Omron Sysmac Studio project RemoteLab (Sysmac Studio 1.47.0.64008, StandardProject)

# Controller Controller_0: NJ301-1100 version 1.20
Units and slaves: Power Supply : NJ-Px3001; CPU : NJ301-1100; 0 : CJ1W-ID211 (J01); 1 : CJ1W-OC211 (J02)
Task PrimaryTask (priority 4, period or condition 4000): PrimaryTask_Main
Task CommTask (priority 16, period or condition 100000): CommTask_ModbusServer
Task ControlTask (priority 16, period or condition 40000): ControlTask_PID
Library MTCP_Server_NJNX 2.6. (contents left out)
Library MTCP_Client_NJ 2.6. (contents left out)

VAR_GLOBAL
    G_Eff_Mode : INT;
    G_Eff_PLC_Enable : BOOL;
    G_Eff_Setpoint : REAL;
    G_Eff_Manual_MV : REAL;
    G_Eff_StartAT : BOOL;
    G_Modbus_ReadBuf : ARRAY[0..1023] OF WORD;  (* Raw Read Data *)
    G_Modbus_WriteBuf : ARRAY[0..1023] OF WORD;  (* Raw Write Data (Mirror of Gateway HRs) *)
    G_OverheatLatched : BOOL;
    StartServer : BOOL := True;
    G_RTD_Temp : REAL;
    G_Setpoint : REAL := 0.0;
    G_StartAT : INT := 0;
    G_ATDone : WORD;
    G_Web_Status : INT := 0;  (* written by CommTask from HR3 *)
    G_Current_MV : REAL;
    G_Manual_MV : REAL := 0.0;  (* Extracted Manual MV *)
    G_Mode : INT := 0;  (* 0=Manual, 1=Auto, 2=Tune *)
    G_PID_PB : REAL;
END_VAR
VAR_GLOBAL RETAIN
    G_PID_PB_Out : REAL := 8.8;
END_VAR
VAR_GLOBAL
    G_PID_Td : REAL;
END_VAR
VAR_GLOBAL RETAIN
    G_PID_Td_Out : REAL := 50;
END_VAR
VAR_GLOBAL
    G_PID_Ti : REAL;
    HMI_AT_ON_Rise : BOOL;
    HMI_AT_OFF_Rise : BOOL;
    HMI_AT_ON_Prev : BOOL;
    HMI_AT_OFF_Prev : BOOL;
END_VAR
VAR_GLOBAL RETAIN
    G_PID_Ti_Out : REAL := 140;
END_VAR
VAR_GLOBAL
    G_PLC_Status : INT := 0;
    Heartbeat_Ctr : UINT;
    G_CommAlive : BOOL;  (* written by PrimaryTask (watchdog) *)
    HMI_Mode : INT;
    HMI_PLC_Enable : BOOL;  (* Momentary button to apply changes *)
    HMI_Setpoint : REAL;
    HMI_Manual_MV : REAL;
    HMI_AT_ON : BOOL;  (* Momentary pushbutton — Start Auto-Tune *)
    HMI_AT_OFF : BOOL;  (* Momentary pushbutton — Stop Auto-Tune *)
    HMI_StartAT : BOOL;
    Out_0 : BOOL;  (* Green LED; at IOBus://rack#0/slot#1/Ch1_Out/Ch1_Out00 *)
    Out_1 : BOOL;  (* Yellow LED; at IOBus://rack#0/slot#1/Ch1_Out/Ch1_Out01 *)
    Out_2 : BOOL;  (* RED LED; at IOBus://rack#0/slot#1/Ch1_Out/Ch1_Out02 *)
    Out_3 : BOOL;  (* PWM output to heater driver; at IOBus://rack#0/slot#1/Ch1_Out/Ch1_Out03 *)
    G_ATBusy : WORD;
    G_Tune_Err : WORD;
    G_WebActive : BOOL;
    HMI_PID_PB : REAL;  (* Proportional Band *)
    HMI_PID_Ti : REAL;  (* Integral Time (seconds) *)
    HMI_PID_Td : REAL;  (* Derivative Time (seconds) *)
    HMI_PID_Update : BOOL;
    HMI_PID_Update_Rise : BOOL;
    HMI_PID_Update_Prev : BOOL;
    HMI_PID_Update_Feedback : BOOL;  (* momentary indicator that tells the operator "Your parameters were successfully applied!" *)
    G_Eff_PID_PB : REAL;
    G_Eff_PID_Ti : REAL;
    G_Eff_PID_Td : REAL;
    C_MODE_MANUAL : INT := 0;
    C_MODE_AUTO : INT := 1;
    C_MODE_TUNE : INT := 2;
    HMI_Manual_MV_DataEdit : REAL;
    HMI_Setpoint_DataEdit : REAL;
    G_Mode_Manual : BOOL;
    G_Mode_AT : BOOL;
    G_Mode_Auto : BOOL;
    HMI_Manual_Start_Rise : BOOL;
    HMI_Manual_Start_Prev : BOOL;
    HMI_Manual_Start : BOOL;
    HMI_Manual_Stop : BOOL;
    HMI_Manual_Stop_Rise : BOOL;
    HMI_Manual_Stop_Prev : BOOL;
    G_PID_PB_AT : REAL;
    G_PID_Ti_AT : REAL;
    G_PID_Td_AT : REAL;
    HMI_Automatic_Start : BOOL;
    HMI_Automatic_Start_Rise : BOOL;
    HMI_Automatic_Start_Prev : BOOL;
    HMI_Automatic_Stop : BOOL;
    HMI_Automatic_Stop_Rise : BOOL;
    HMI_Automatic_Stop_Prev : BOOL;
    G_Heater_Power_W : REAL;
    G_ATDone_FB : BOOL;
END_VAR

PROGRAM CommTask_ModbusServer
VAR
    MB_Server : MTCP_Server_NJNX;
    Local_TcpPort : UINT := 1502;
    ConnectionTimeout : TIME := T#0ms;
    Reset_SdRcvCounter : BOOL := False;
    Server_Connected : BOOL;
    Server_Error : BOOL;
    Server_ErrorID : WORD;
    IP_Client : STRING[15];
    Port_Client : UINT;
    SdRcv_Counter : UDINT;
    SdRcv_Last : UDINT;
    Coils : ARRAY[0..1023] OF BOOL;
    Registers : ARRAY[0..1023] OF WORD;
    i : INT;
    New_Seq : WORD;
    Last_Seq_Num : WORD;
    R2W_MV : FB_RealToWords;
    R2W_PB : FB_RealToWords;
    R2W_Ti : FB_RealToWords;
    R2W_Td : FB_RealToWords;
    R2W_Setpoint : FB_RealToWords;
    R2W_PB_AT : FB_RealToWords;
    R2W_Ti_AT : FB_RealToWords;
    R2W_Td_AT : FB_RealToWords;
END_VAR
VAR_EXTERNAL
    G_Modbus_ReadBuf : ARRAY[0..1023] OF WORD;
    StartServer : BOOL;
    G_Web_Status : INT;
    G_Mode : INT;
    G_PLC_Status : INT;
    G_Manual_MV : REAL;
    G_Setpoint : REAL;
    G_StartAT : INT;
    G_PID_PB : REAL;
    G_PID_Ti : REAL;
    G_PID_Td : REAL;
    G_Current_MV : REAL;
    G_PID_Td_Out : REAL;
    G_Modbus_WriteBuf : ARRAY[0..1023] OF WORD;
    G_RTD_Temp : REAL;
    G_PID_PB_Out : REAL;
    G_PID_Ti_Out : REAL;
    Heartbeat_Ctr : UINT;
    G_ATDone : WORD;
    G_Eff_Setpoint : REAL;
    G_PID_PB_AT : REAL;
    G_PID_Ti_AT : REAL;
    G_PID_Td_AT : REAL;
    G_ATBusy : WORD;
    G_ATDone_FB : BOOL;
    G_Tune_Err : WORD;
END_VAR
(*
    CommTask_ModbusServer
    - PLC is Modbus TCP SERVER (slave)
    - Gateway/Web is Modbus TCP CLIENT (master)
*)

// =========================================================
// 1) Run the Modbus TCP Server FB EVERY scan
// =========================================================
MB_Server(
    Start             := StartServer,
    Local_TcpPort     := Local_TcpPort,
    ConnectionTimeout := ConnectionTimeout,
    Reset_SdRcvCounter:= Reset_SdRcvCounter,

    Registers         := Registers,
    Coils             := Coils,

    Connected         => Server_Connected,
    Error             => Server_Error,
    ErrorID           => Server_ErrorID,
    IP_Client         => IP_Client,
    Port_Client       => Port_Client,
    SdRcv_Counter     => SdRcv_Counter
);


// =========================================================
// 2) Heartbeat: increment when a Modbus transaction happened
//    (so it tracks real comm activity)
// =========================================================
IF SdRcv_Counter <> SdRcv_Last THEN
    SdRcv_Last := SdRcv_Counter;
    Heartbeat_Ctr := Heartbeat_Ctr + 1;
END_IF;


// =========================================================
// 3) Copy incoming gateway-written registers into your buffer
//    (HR0..HR16 -> G_Modbus_ReadBuf[0..16])
// =========================================================
FOR i := 0 TO 16 DO
    G_Modbus_ReadBuf[i] := Registers[i];
END_FOR;


// =========================================================
// 4) PROCESS (same as your old State 20)
// =========================================================
G_RTD_Temp := FUN_WordsToReal(G_Modbus_ReadBuf[1], G_Modbus_ReadBuf[2]);

New_Seq := G_Modbus_ReadBuf[0];

IF New_Seq <> Last_Seq_Num THEN
    G_Web_Status := WORD_TO_INT(G_Modbus_ReadBuf[3]);
    G_Mode       := WORD_TO_INT(G_Modbus_ReadBuf[4]);
    G_PLC_Status := WORD_TO_INT(G_Modbus_ReadBuf[5]);

    G_Manual_MV  := FUN_WordsToReal(G_Modbus_ReadBuf[6], G_Modbus_ReadBuf[7]);
    G_Setpoint   := FUN_WordsToReal(G_Modbus_ReadBuf[8], G_Modbus_ReadBuf[9]);

    G_StartAT   := WORD_TO_INT(G_Modbus_ReadBuf[10]);

    G_PID_PB     := FUN_WordsToReal(G_Modbus_ReadBuf[11], G_Modbus_ReadBuf[12]);
    G_PID_Ti     := FUN_WordsToReal(G_Modbus_ReadBuf[13], G_Modbus_ReadBuf[14]);
    G_PID_Td     := FUN_WordsToReal(G_Modbus_ReadBuf[15], G_Modbus_ReadBuf[16]);

    Last_Seq_Num := New_Seq;
END_IF;


// =========================================================
// 5) BUILD WRITE BUFFER (same as your old State 30)
//    (HR100..HR110 -> G_Modbus_WriteBuf[0..10])
// =========================================================
G_Modbus_WriteBuf[0] := Last_Seq_Num;                // HR100 ack seq
G_Modbus_WriteBuf[1] := UINT_TO_WORD(Heartbeat_Ctr); // HR101 heartbeat

R2W_MV(InReal := G_Current_MV);
G_Modbus_WriteBuf[2] := R2W_MV.W_High;               // HR102  -- Current_MV
G_Modbus_WriteBuf[3] := R2W_MV.W_Low;                // HR103

// ===== Autotune Status =====
G_Modbus_WriteBuf[4] := G_ATBusy;        // HR104  autotune running
G_Modbus_WriteBuf[5] := G_ATDone;     // HR105  autotune finished
G_Modbus_WriteBuf[6] := G_Tune_Err;      // HR106  autotune error

// ===== Current PID parameters =====
R2W_PB(InReal := G_PID_PB_Out);
G_Modbus_WriteBuf[7] := R2W_PB.W_High;               // HR107
G_Modbus_WriteBuf[8] := R2W_PB.W_Low;                // HR108

R2W_Ti(InReal := G_PID_Ti_Out);
G_Modbus_WriteBuf[9]  := R2W_Ti.W_High;              // HR109
G_Modbus_WriteBuf[10] := R2W_Ti.W_Low;               // HR110

R2W_Td(InReal := G_PID_Td_Out);
G_Modbus_WriteBuf[11] := R2W_Td.W_High;              // HR111
G_Modbus_WriteBuf[12] := R2W_Td.W_Low;               // HR112

// ===== Current Setpoint =====
R2W_Setpoint(InReal := G_Eff_Setpoint);
G_Modbus_WriteBuf[13] := R2W_Setpoint.W_High;        // HR113
G_Modbus_WriteBuf[14] := R2W_Setpoint.W_Low;         // HR114

// ===== Autotune Results =====
R2W_PB_AT(InReal := G_PID_PB_AT);
G_Modbus_WriteBuf[15] := R2W_PB_AT.W_High;           // HR115
G_Modbus_WriteBuf[16] := R2W_PB_AT.W_Low;            // HR116

R2W_Ti_AT(InReal := G_PID_Ti_AT);
G_Modbus_WriteBuf[17] := R2W_Ti_AT.W_High;           // HR117
G_Modbus_WriteBuf[18] := R2W_Ti_AT.W_Low;            // HR118

R2W_Td_AT(InReal := G_PID_Td_AT);
G_Modbus_WriteBuf[19] := R2W_Td_AT.W_High;           // HR119
G_Modbus_WriteBuf[20] := R2W_Td_AT.W_Low;            // HR120

// =========================================================
// 6) Copy your write buffer into server registers
//    (G_Modbus_WriteBuf -> HR100..HR110)
// =========================================================
FOR i := 0 TO 20 DO
    Registers[100 + i] := G_Modbus_WriteBuf[i];
END_FOR;
END_PROGRAM

PROGRAM ControlTask_PID
VAR
    ATBusy_FB : BOOL;
    ATErr_FB : BOOL;
    ATErrID_FB : WORD;
    TuneCmd : BOOL;
    Ti_ms : DINT;
    Td_ms : DINT;
    Ti_Time : TIME;
    Td_Time : TIME;
    StartAT_Cmd : BOOL;
    RunCmd : BOOL;
    MV_fromPID : REAL;
    MV_percent : REAL;
    OprSetParams : _sOPR_SET_PARAMS := (MVLowLmt := 0.0, MVUpLmt := 100.0, ManResetVal := 0.0, MVTrackSw := False, MVTrackVal := 0.0, StopMV := 0.0, ErrorMV := 0.0, Alpha := 0.0, ATCalcGain := 1.0, ATHystrs := 0.2);
    InitSetParams : _sINIT_SET_PARAMS := (SampTime := T#200mS, RngLowLmt := 0.0, RngUpLmt := 150.0, DirOpr := False);
    PB_Active : REAL;
    Ti_Active_s : REAL;
    Td_Active_s : REAL;
    Ti_Active : REAL;
    Td_Active : REAL;
    PIDAT_instance : PIDAT;
    ATDone_Rise : BOOL;
    ATDone_Prev : BOOL;
END_VAR
VAR_EXTERNAL
    G_Eff_Mode : INT;
    G_PID_PB : REAL;
    G_PID_Ti : REAL;
    G_PID_Td : REAL;
    G_PID_PB_Out : REAL;
    G_PID_Ti_Out : REAL;
    G_PID_Td_Out : REAL;
    G_Eff_PLC_Enable : BOOL;
    G_OverheatLatched : BOOL;
    G_Eff_StartAT : BOOL;
    G_RTD_Temp : REAL;
    G_Eff_Setpoint : REAL;
    G_Eff_Manual_MV : REAL;
    G_Current_MV : REAL;
    G_ATBusy : WORD;
    G_Tune_Err : WORD;
    G_ATDone : WORD;
    G_WebActive : BOOL;
    HMI_PID_PB : REAL;
    HMI_PID_Ti : REAL;
    HMI_PID_Td : REAL;
    HMI_PID_Update_Rise : BOOL;
    HMI_PID_Update : BOOL;
    HMI_PID_Update_Prev : BOOL;
    HMI_PID_Update_Feedback : BOOL;
    G_Eff_PID_PB : REAL;
    G_Eff_PID_Ti : REAL;
    G_Eff_PID_Td : REAL;
    C_MODE_MANUAL : INT;
    C_MODE_AUTO : INT;
    C_MODE_TUNE : INT;
    G_Mode_Manual : BOOL;
    G_Mode_AT : BOOL;
    G_ATDone_FB : BOOL;
    G_PID_PB_AT : REAL;
    G_PID_Ti_AT : REAL;
    G_PID_Td_AT : REAL;
    G_StartAT : INT;
    HMI_StartAT : BOOL;
END_VAR
(*
    ControlTask_PID
    - With HMI_PID_Update apply button
    - 
*)


// ---------------------------------------------------------
// 2) Run condition (already selected Web/Local in PrimaryTask)
// ---------------------------------------------------------
RunCmd := G_Eff_PLC_Enable AND (NOT G_OverheatLatched);

// ---------------------------------------------------------
// 3) PID parameter source (REAL seconds stored for web/modbus)
// ---------------------------------------------------------
PB_Active   := G_Eff_PID_PB;
Ti_Active_s := G_Eff_PID_Ti;
Td_Active_s := G_Eff_PID_Td;

// ---------------------------------------------------------
// 3b) Convert REAL seconds -> TIME (milliseconds resolution)
// ---------------------------------------------------------
// Ti_Active_s, Td_Active_s are REAL seconds (from dashboard)
IF Ti_Active_s < 0.0 THEN Ti_Active_s := 0.0; END_IF;
IF Ti_Active_s > 10000.0 THEN Ti_Active_s := 10000.0; END_IF;

IF Td_Active_s < 0.0 THEN Td_Active_s := 0.0; END_IF;
IF Td_Active_s > 10000.0 THEN Td_Active_s := 10000.0; END_IF;

// REAL seconds -> TIME (seconds resolution)
Ti_Time := SecToTime( REAL_TO_LINT(Ti_Active_s + 0.5) );
Td_Time := SecToTime( REAL_TO_LINT(Td_Active_s + 0.5) );


// ---------------------------------------------------------
// 4) Call PIDAT (40ms task = good for thermal control)
//    IMPORTANT: set OprSetParams cycle time = 40ms in your init/vars
// ---------------------------------------------------------
PIDAT_instance(
    Run            := RunCmd,
    ManCtl         := G_Mode_Manual,          // TRUE=manual, FALSE=auto/tune
    StartAT        := G_Eff_StartAT,
    PV             := G_RTD_Temp,
    SP             := G_Eff_Setpoint,
    OprSetParams   := OprSetParams,        // your struct
    InitSetParams  := InitSetParams,       // your struct (InitType can be tied to mode if you want)
    ProportionalBand := PB_Active,
    IntegrationTime  := Ti_Time,
    DerivativeTime   := Td_Time,
    ManMV          := G_Eff_Manual_MV,	
	ATDone  => G_ATDone_FB,
    ATBusy  => ATBusy_FB,
    Error   => ATErr_FB,
    ErrorID => ATErrID_FB,
    MV      => MV_fromPID
);

// ---------------------------------------------------------
// 5) Decide the final MV (single source of truth)
// ---------------------------------------------------------
IF NOT RunCmd THEN
    G_Current_MV := 0.0;
ELSE
    IF G_Mode_Manual THEN
        G_Current_MV := G_Eff_Manual_MV;
    ELSE
        G_Current_MV := MV_fromPID;
    END_IF;
END_IF;
// ---------------------------------------------------------
// 6) Detect autotune completion
// ---------------------------------------------------------
ATDone_Rise := G_ATDone_FB AND NOT ATDone_Prev;
ATDone_Prev := G_ATDone_FB;

IF ATDone_Rise THEN

    // Capture tuned parameters
    G_PID_PB_AT := PB_Active;
	
    // Convert TIME -> REAL seconds
    G_PID_Ti_AT := LINT_TO_REAL(TimeToSec(In := Ti_Time));
    G_PID_Td_AT := LINT_TO_REAL(TimeToSec(In := Td_Time));

    // Reset autotune command
    IF G_WebActive THEN
        G_StartAT := 0;
    ELSE
        HMI_StartAT := FALSE;
    END_IF;
END_IF;

// ---------------------------------------------------------
// 7) Report current active PID to web
// ---------------------------------------------------------
G_PID_PB_Out := G_Eff_PID_PB;
G_PID_Ti_Out := G_Eff_PID_Ti;
G_PID_Td_Out := G_Eff_PID_Td;


IF ATBusy_FB THEN G_ATBusy := WORD#1; ELSE G_ATBusy := WORD#0; END_IF;
IF ATErr_FB  THEN G_Tune_Err  := WORD#1; ELSE G_Tune_Err  := WORD#0; END_IF;
IF G_ATDone_FB THEN  G_ATDone := WORD#1;ELSE  G_ATDone := WORD#0; END_IF;
END_PROGRAM

PROGRAM PrimaryTask_Main
VAR
    HB_Last : UINT;
    CommWd : TON;
    FirstScanDone : BOOL := False;
    TempOver : BOOL;
    WebPrev : BOOL;
    WebRise : BOOL;
    ResetArmed : BOOL;
    MV_percent : REAL;
    PWM_Out : TimeProportionalOut;
    MV_Limited : REAL;
    PWM_Enable : BOOL;
END_VAR
VAR_EXTERNAL
    Heartbeat_Ctr : UINT;
    G_Mode : INT;
    G_PLC_Status : INT;
    G_Setpoint : REAL;
    G_Manual_MV : REAL;
    G_StartAT : INT;
    G_CommAlive : BOOL;
    G_Eff_Mode : INT;
    G_Eff_Setpoint : REAL;
    G_Eff_Manual_MV : REAL;
    HMI_Mode : INT;
    HMI_StartAT : BOOL;
    HMI_Manual_MV : REAL;
    HMI_Setpoint : REAL;
    HMI_PLC_Enable : BOOL;
    G_Eff_StartAT : BOOL;
    G_RTD_Temp : REAL;
    G_Web_Status : INT;
    G_OverheatLatched : BOOL;
    G_Eff_PLC_Enable : BOOL;
    Out_3 : BOOL;
    Out_2 : BOOL;
    Out_1 : BOOL;
    Out_0 : BOOL;
    G_WebActive : BOOL;
    G_Eff_PID_PB : REAL;
    G_PID_PB : REAL;
    G_Eff_PID_Ti : REAL;
    G_Eff_PID_Td : REAL;
    G_PID_Ti : REAL;
    G_PID_Td : REAL;
    HMI_PID_Update_Rise : BOOL;
    HMI_PID_Update : BOOL;
    HMI_PID_Update_Prev : BOOL;
    HMI_PID_Update_Feedback : BOOL;
    HMI_PID_PB : REAL;
    HMI_PID_Ti : REAL;
    HMI_PID_Td : REAL;
    G_PID_PB_Out : REAL;
    G_PID_Ti_Out : REAL;
    G_PID_Td_Out : REAL;
    C_MODE_MANUAL : INT;
    C_MODE_AUTO : INT;
    C_MODE_TUNE : INT;
    G_Current_MV : REAL;
    HMI_AT_ON : BOOL;
    HMI_AT_OFF : BOOL;
    HMI_AT_ON_Rise : BOOL;
    HMI_AT_OFF_Rise : BOOL;
    HMI_AT_ON_Prev : BOOL;
    HMI_AT_OFF_Prev : BOOL;
    G_Mode_Manual : BOOL;
    G_Mode_AT : BOOL;
    G_Mode_Auto : BOOL;
    HMI_Manual_Start_Rise : BOOL;
    HMI_Manual_Stop_Rise : BOOL;
    HMI_Manual_Start_Prev : BOOL;
    HMI_Manual_Stop_Prev : BOOL;
    HMI_Automatic_Stop_Rise : BOOL;
    HMI_Automatic_Start_Rise : BOOL;
    HMI_Automatic_Start_Prev : BOOL;
    HMI_Manual_Start : BOOL;
    HMI_Manual_Stop : BOOL;
    HMI_Automatic_Stop_Prev : BOOL;
    HMI_Automatic_Start : BOOL;
    HMI_Automatic_Stop : BOOL;
    HMI_Setpoint_DataEdit : REAL;
    HMI_Manual_MV_DataEdit : REAL;
    G_Heater_Power_W : REAL;
END_VAR
(*
    PrimaryTask+Main
	- G_PID_* → web buffer (read from the modbus HR)
	- G_Eff_PID_* → used by ControlTask
	- HMI_PID_* → operator entry values
	- G_PID_*_Out → actual running PID parameters (write to the modbus HR)
    - 
*)

G_Mode_Manual := (G_Eff_Mode = C_MODE_MANUAL);
G_Mode_Auto     := (G_Eff_Mode = C_MODE_AUTO);
G_Mode_AT         := (G_Eff_Mode = C_MODE_TUNE);

// First scan initialization
IF NOT FirstScanDone THEN
    // === First Scan Initialization ===
    G_Eff_PID_PB := G_PID_PB_Out;
    G_Eff_PID_Ti := G_PID_Ti_Out;
    G_Eff_PID_Td := G_PID_Td_Out;
    FirstScanDone := TRUE;
END_IF;

// ---------------------------------------------------------
// 0) COMM ALIVE watchdog (uses your Heartbeat_Ctr that increments on Modbus traffic)
// I (PLC) am confident comms are alive, so web takeover is allowed?
// this is to prevent the PLC won’t stay stuck in “web owns control” forever.
// ---------------------------------------------------------
IF Heartbeat_Ctr <> HB_Last THEN
    HB_Last := Heartbeat_Ctr;
    CommWd(IN := FALSE); // reset TON
END_IF;

CommWd(IN := TRUE, PT := T#2s);
G_CommAlive := NOT CommWd.Q;

// ---------------------------------------------------------
// 1) Edge detection for HMI_PID_Update (add this)
// ---------------------------------------------------------
HMI_PID_Update_Rise := (HMI_PID_Update AND NOT HMI_PID_Update_Prev);
HMI_PID_Update_Prev := HMI_PID_Update;

// ---------------------------------------------------------
// 1b) HMI_PLC_Enable Button Edge Detection
// ---------------------------------------------------------
HMI_Manual_Start_Rise := (HMI_Manual_Start AND NOT HMI_Manual_Start_Prev);
HMI_Manual_Stop_Rise  := (HMI_Manual_Stop  AND NOT HMI_Manual_Stop_Prev);

HMI_Manual_Start_Prev := HMI_Manual_Start;
HMI_Manual_Stop_Prev  := HMI_Manual_Stop;

HMI_Automatic_Start_Rise := (HMI_Automatic_Start AND NOT HMI_Automatic_Start_Prev);
HMI_Automatic_Stop_Rise  := (HMI_Automatic_Stop  AND NOT HMI_Automatic_Stop_Prev);

HMI_Automatic_Start_Prev := HMI_Automatic_Start;
HMI_Automatic_Stop_Prev  := HMI_Automatic_Stop;


// ---------------------------------------------------------
// 1c) HMI Auto-Tune Button Edge Detection
// ---------------------------------------------------------
HMI_AT_ON_Rise  := (HMI_AT_ON AND NOT HMI_AT_ON_Prev);
HMI_AT_OFF_Rise := (HMI_AT_OFF AND NOT HMI_AT_OFF_Prev);

HMI_AT_ON_Prev  := HMI_AT_ON;
HMI_AT_OFF_Prev := HMI_AT_OFF;

// ---------------------------------------------------------
// 2) Web takeover decision (require comm alive if Web wants control)
// ---------------------------------------------------------
G_WebActive := (G_Web_Status <> 0) AND G_CommAlive;

// ---------------------------------------------------------
// 3a) Select EFFECTIVE commands (Web vs Local HMI)
// - Continuous scan reading when G_WebActive is TRUE
// ---------------------------------------------------------
IF G_WebActive THEN
    G_Eff_Mode          := G_Mode;
    G_Eff_PLC_Enable := (G_PLC_Status <> 0);
    G_Eff_Setpoint      := G_Setpoint;
    G_Eff_Manual_MV := G_Manual_MV;
    G_Eff_StartAT    := (G_StartAT <> 0);
ELSE
    // Local / NA5 takeover when Web is off
    G_Eff_Mode       := HMI_Mode;
    G_Eff_PLC_Enable := HMI_PLC_Enable;
    G_Eff_Setpoint   := HMI_Setpoint;
    G_Eff_Manual_MV  := HMI_Manual_MV;
    G_Eff_StartAT    := HMI_StartAT;
END_IF;

// ---------------------------------------------------------
// 3 b) HMI: latch ONLY on Apply button rising edge
// ---------------------------------------------------------
IF G_WebActive THEN
	G_Eff_PID_PB        := G_PID_PB;
    G_Eff_PID_Ti         := G_PID_Ti;
    G_Eff_PID_Td        := G_PID_Td;
ELSIF HMI_PID_Update_Rise THEN 	
    // HMI can adjust PID parameters - only on Apply button click
    G_Eff_PID_PB     := HMI_PID_PB;      // Copy HMI -> Web buffer
    G_Eff_PID_Ti      := HMI_PID_Ti;
    G_Eff_PID_Td     := HMI_PID_Td;
    
    // Optional: Provide feedback that parameters were applied
    HMI_PID_Update_Feedback := TRUE;  // flash confirmation on NA page
END_IF;
// If neither: EFF_PID_* retains its last value → built-in latch!

// Clear feedback next scan
IF NOT HMI_PID_Update_Rise THEN
    HMI_PID_Update_Feedback := FALSE;
END_IF;

// ---------------------------------------------------------
// 3c) HMI PLC_Enable  Latch Logic
// ---------------------------------------------------------
IF HMI_Manual_Start_Rise THEN
	HMI_Mode :=C_MODE_MANUAL;
    HMI_PLC_Enable := TRUE;
END_IF;

IF HMI_Manual_Stop_Rise THEN
    HMI_PLC_Enable := FALSE;
END_IF;

IF HMI_Automatic_Start_Rise THEN
	HMI_Mode := C_MODE_AUTO;
    HMI_PLC_Enable := TRUE;
END_IF;

IF HMI_Automatic_Stop_Rise THEN
    HMI_PLC_Enable := FALSE;
END_IF;
// ---------------------------------------------------------
// 3d) HMI Auto-Tune Latch Logic
// ---------------------------------------------------------
// Start tuning
IF HMI_AT_ON_Rise THEN
    HMI_StartAT := TRUE;
END_IF;

// Stop tuning (operator interrupt)
IF HMI_AT_OFF_Rise THEN
    HMI_StartAT := FALSE;
END_IF;


// ---------------------------------------------------------
// 4) Overheat latch (Trip at >100C, require Web OFF->ON to reset)
// ---------------------------------------------------------
TempOver := (G_RTD_Temp > 100.0);

IF TempOver THEN
    G_OverheatLatched := TRUE;
END_IF;

// Rising edge detect of raw Web command (not G_WebActive)
WebRise := ( (G_Web_Status <> 0) AND (NOT WebPrev) );
WebPrev := (G_Web_Status <> 0);

// Arm reset when Web is OFF
IF (G_Web_Status = 0) THEN
    ResetArmed := TRUE;
END_IF;

// Clear latch only when Web toggles OFF then ON
IF WebRise AND ResetArmed THEN
    G_OverheatLatched := FALSE;
    ResetArmed := FALSE;
END_IF;
// ---------------------------------------------------------
// 5) Final output gating + PWM (using G_Current_MV directly)
// ---------------------------------------------------------
IF (NOT G_Eff_PLC_Enable) OR G_OverheatLatched THEN
    MV_Limited := 0.0;
ELSE
    // Use G_Current_MV directly from ControlTask
    IF G_Current_MV < 0.0 THEN MV_Limited := 0.0;
    ELSIF G_Current_MV > 100.0 THEN MV_Limited := 100.0;
    ELSE MV_Limited := G_Current_MV;
    END_IF;
END_IF;

G_Heater_Power_W := (MV_Limited / 100.0) * 11.52;

// Call your TimeProportionalOut FB every 4ms for clean timing
PWM_Enable := G_Eff_PLC_Enable AND NOT G_OverheatLatched;
PWM_Out(
	Enable:=PWM_Enable,
    Ain     := MV_Limited,     // adjust input name if different in your FB
    CtlPrd := T#1s,
	MinPlsWidth :=0.0,
	Delay:=0.0,
    DOut   => Out_3
);

// Absolute safety override (belt + braces)
IF G_OverheatLatched THEN
    Out_3 := FALSE;
END_IF;

// ---------------------------------------------------------
// Stack lights logic (Mode-based)
// ---------------------------------------------------------
Out_0 := (G_Mode_Manual AND G_Eff_PLC_Enable AND NOT G_OverheatLatched);
Out_1 := (G_Mode_Auto   AND G_Eff_PLC_Enable AND NOT G_OverheatLatched);
Out_2 := (G_Mode_AT   AND G_Eff_PLC_Enable AND NOT G_OverheatLatched);
END_PROGRAM

FUNCTION FUN_WordsToReal : REAL
VAR
    TempDWord : DWORD;
END_VAR
VAR_INPUT
    W_High : WORD;
    W_Low : WORD;
END_VAR
(* Combine High and Low words into a DWORD *)
(* Assuming Big Endian Transmission: High Word comes first *)
(* Method: Shift High Word left 16 bits, OR with Low Word *)
TempDWord := SHL(WORD_TO_DWORD(W_High), 16) OR WORD_TO_DWORD(W_Low);

(* Convert bit-wise to REAL (Re-interpret cast) *)
(* In Omron NJ, use the Bit conversion functions if available, or Pointers *)
(* Safest generic way: *)
FUN_WordsToReal := CopyDwordToReal(TempDWord);
END_FUNCTION

FUNCTION_BLOCK FB_RealToWords
VAR
    TempDWord : DWORD;
END_VAR
VAR_INPUT
    InReal : REAL;
END_VAR
VAR_OUTPUT
    W_High : WORD;
    W_Low : WORD;
END_VAR
(* Copy IEEE754 bits of REAL into DWORD *)
TempDWord := CopyRealToDword(In := InReal);

(* Split into High/Low WORD (Big Endian: High first) *)
W_High := TO_WORD(SHR(TempDWord, 16));
W_Low  := TO_WORD(TempDWord);
END_FUNCTION_BLOCK

# Device HMI_0 (NA): not converted